TYPE
    stPositionCommand :
    STRUCT
        Xaxis_Pos : LREAL; // Robot X-axis position command
        Yaxis_Pos : LREAL; // Robot Y-axis position command
        Raxis_Pos : LREAL; // Robot R-axis Position command
    END_STRUCT
END_TYPE

(* stored: Version 1.1.0.1, ProductVersion 3.1.4024.13
   DUT stPositionCommand: Id {92415fc6-3f99-45f6-bda6-8b112f89d8bd} *)
